// TIA Portal V20 export
TYPE "ManualInputs"
// stored: Access Published, Namespace Global
   STRUCT
      ManualEnable : Bool;
      Run : Struct
         Forward : Bool;
         Reverse : Bool;
      END_STRUCT;
   END_STRUCT;
END_TYPE
